Staubli VAL3: mnuTeachPark.pgx

program mnuTeachPark()
  local bool LbBackup
  local num nKey
begin
  //header begin
  // PROGRAM mnuTeachPark()
  //
  // runs the Wizard to assist user:  Teach a single robot PARK position
  // position taught = jPark
  //
  // incoming parms:  none
  // outgoing parms:  none
  // called from:  pgm mnuTeachMenu()
  //
  //  initial release KN
  //header end
  //
  // start continuous loop, go through each of 5 wizard steps
  //
  // init step-by-step continuance booleans
  LbBackup=false
  //
  do
    // nIdxTeachPARK=51
    call displayMessage(nIdxTeachPARK,nKey)
    // verify selection
    switch nKey
      // ESC key aborts & returns immediately
      case 255
        return
      break
      // menu = Teach Park, F1 to continue to Step 2 of 4
      case 271
        jPark=herej()
        LbBackup=true
      break
      // menu = Teach Park, F8 Button, abort to Teach Menu
      case 278
        return
      break
      // Any other key press
      default
        popUpMsg("BAD SELECTION...press OK")
      break
    endSwitch
  until (false or (LbBackup==true))
  //
  // teach Park Position completed, save data on exit
  libSave()
  //
  // done
end
